FUNCTION TFPackCodePresentToJollyWorkArea : INT
VAR_INPUT
	HandlingPackTable : POINTER TO TFHandlingPackTable;
	WorkArea : POINTER TO ARRAY [1..MAXAREA] OF TFMachinePalletizer_WorkArea;
	WorkAreaState : POINTER TO ARRAY [1..MAXAREA] OF TFMachinePalletizer_WorkAreaState;
END_VAR
VAR
	w : INT;
	wa : INT;
	i : INT;
END_VAR

TFPackCodePresentToJollyWorkArea := 0; 

FOR w:=MAXHANDLINGPACK TO 1 BY -1 DO
	IF HandlingPackTable^.Table[w,1].PC > 0 THEN
		FOR wa:=1 TO MAXAREA DO
			IF WorkArea^[wa].Code = HandlingPackTable^.Table[w,1].PC THEN
				(* Verifico se la piazzola è in lavorazione *)
				(* Se è in lavorazione allora è inutile assegnarne un'altra con lo stesso codice *)
				IF WorkAreaState^[wa].State < WORKAREA_STATE_OCCUPIED_WORKED THEN
					TFPackCodePresentToJollyWorkArea := 0;
					RETURN;
				//ELSE
					//TFPackCodePresentToJollyWorkArea := WorkPickPointState^[w].Code;
				END_IF
				//RETURN;
			END_IF
		END_FOR
		TFPackCodePresentToJollyWorkArea := HandlingPackTable^.Table[w,1].PC;
	END_IF	
END_FOR

END_FUNCTION

(* stored: Version 1.1.0.1, ProductVersion 3.1.4024.11
   POU TFPackCodePresentToJollyWorkArea: Id {1be65bd6-ee28-46f1-ba60-40b04d45a60e}, SpecialFunc None *)
